% RSLogix 500 project PLC Level 2 Project 3.RSS, saved by version 8.30.00.16 %
PROJECT "UNTITLED"    % processor: Bul.1763 MicroLogix 1100 Series B %

PROGRAM FILES
  LAD 2 "MAIN"  5 rungs

DATA FILES
  O0 OUTPUT  4 elements
  I1 INPUT  6 elements
  S2 STATUS  66 elements
  B3 BINARY  1 elements
  T4 TIMER  1 elements
  C5 COUNTER  1 elements
  R6 CONTROL  1 elements
  N7 INTEGER  9 elements
  F8 FLOAT  1 elements
  ST9 STRING  11 elements

LADDER 2 "MAIN"
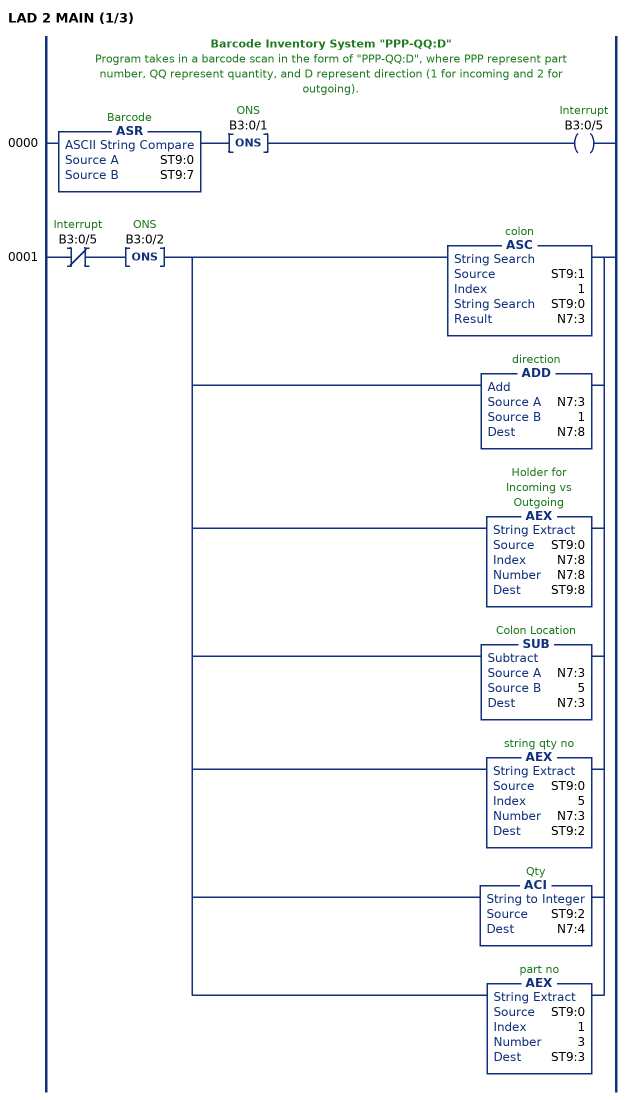
% Rung: 0 %
% TITLE: Barcode Inventory System "PPP-QQ:D" %
% Program takes in a barcode scan in the form of "PPP-QQ:D", where PPP represent part number, QQ represent quantity, and D represent direction (1 for incoming and 2 for outgoing). %
SOR ASR ST9:0 ST9:7 ONS B3:0/1 OTE B3:0/5 EOR
%   ST9:0  "Barcode" %
%   ST9:7  "blank" %
%   B3:0/1  "ONS" %
%   B3:0/5  "Interrupt" %
% Rung: 1 %
SOR XIO B3:0/5 ONS B3:0/2 BST ASC ST9:1 1 ST9:0 N7:3 NXB ADD N7:3 1 N7:8 NXB AEX ST9:0 N7:8 N7:8 ST9:8 NXB SUB N7:3 5 N7:3 NXB AEX ST9:0 5 N7:3 ST9:2 NXB ACI ST9:2 N7:4 NXB AEX ST9:0 1 3 ST9:3 BND EOR
%   B3:0/5  "Interrupt" %
%   B3:0/2  "ONS" %
%   ST9:1  "colon" %
%   ST9:0  "Barcode" %
%   N7:3  "Colon Location" %
%   N7:8  "direction" %
%   ST9:8  "Holder for Incoming vs Outgoing" %
%   ST9:2  "string qty no" %
%   N7:4  "Qty" %
%   ST9:3  "part no" %

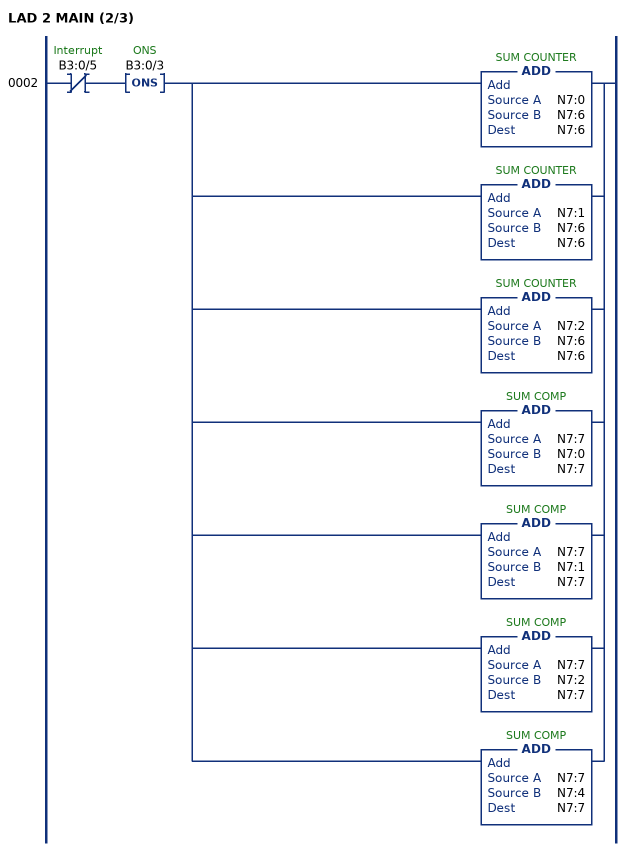
% Rung: 2 %
SOR XIO B3:0/5 ONS B3:0/3 BST ADD N7:0 N7:6 N7:6 NXB ADD N7:1 N7:6 N7:6 NXB ADD N7:2 N7:6 N7:6 NXB ADD N7:7 N7:0 N7:7 NXB ADD N7:7 N7:1 N7:7 NXB ADD N7:7 N7:2 N7:7 NXB ADD N7:7 N7:4 N7:7 BND EOR
%   B3:0/5  "Interrupt" %
%   B3:0/3  "ONS" %
%   N7:0  "Part #123" %
%   N7:6  "SUM COUNTER" %
%   N7:1  "Part #456" %
%   N7:2  "Part #789" %
%   N7:7  "SUM COMP" %
%   N7:4  "Qty" %

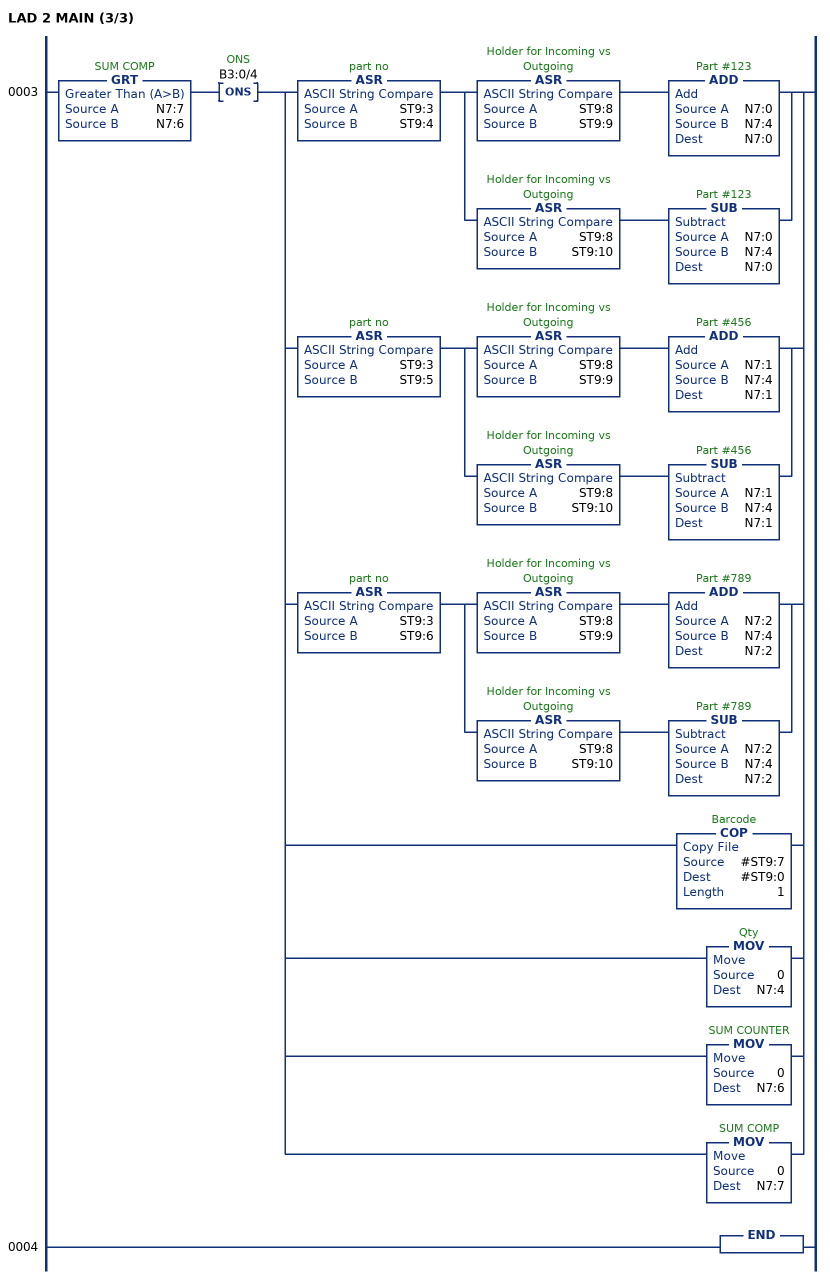
% Rung: 3 %
SOR GRT N7:7 N7:6 ONS B3:0/4 BST ASR ST9:3 ST9:4 BST ASR ST9:8 ST9:9 ADD N7:0 N7:4 N7:0 NXB ASR ST9:8 ST9:10 SUB N7:0 N7:4 N7:0 BND NXB ASR ST9:3 ST9:5 BST ASR ST9:8 ST9:9 ADD N7:1 N7:4 N7:1 NXB ASR ST9:8 ST9:10 SUB N7:1 N7:4 N7:1 BND NXB ASR ST9:3 ST9:6 BST ASR ST9:8 ST9:9 ADD N7:2 N7:4 N7:2 NXB ASR ST9:8 ST9:10 SUB N7:2 N7:4 N7:2 BND NXB COP #ST9:7 #ST9:0 1 NXB MOV 0 N7:4 NXB MOV 0 N7:6 NXB MOV 0 N7:7 BND EOR
%   N7:7  "SUM COMP" %
%   N7:6  "SUM COUNTER" %
%   B3:0/4  "ONS" %
%   ST9:3  "part no" %
%   ST9:4  "part no 123" %
%   ST9:8  "Holder for Incoming vs Outgoing" %
%   ST9:9  "Incoming" %
%   N7:0  "Part #123" %
%   N7:4  "Qty" %
%   ST9:10  "Outgoing" %
%   ST9:5  "part no 456" %
%   N7:1  "Part #456" %
%   ST9:6  "part no 789" %
%   N7:2  "Part #789" %
%   ST9:7  "blank" %
%   ST9:0  "Barcode" %
% Rung: 4 %
SOR END EOR

OTHER DOCUMENTED ADDRESSES
  B3:0/0  "TEST"
  N7:5  "blank"
  ST9:7.0  "blank"
  TEST  
  U:3  "EXTRACT QTY"

DATA TABLE (non-zero values as saved)
DATA ST9
% ST9:1 % ":"
% ST9:4 % "123"
% ST9:5 % "456"
% ST9:6 % "789"
% ST9:9 % "1"
% ST9:10 % "2"
